# EPICS IOC start-up script: iocsh/ethercatmcReleaseBrake.iocsh
ethercatmcCreateAsynParam $(MOTOR_PORT) ReleaseBrake Int32

dbLoadRecords("ethercatmcReleaseBrake.template", "PREFIX=$(PREFIX), AXIS_NAME=$(AXIS_NAME), DESC=$(DESC), MOTOR_PORT=$(MOTOR_PORT), AXIS_NO=$(AXIS_NO)")
